Staubli VAL3: onStop.pgx

public program onStop(string& x_sItem[])
  local num i
begin
  // reset the bit
  for i=0 to size(bExecute)-1
    bExecute[i]=false
  endFor
end
